// List of Strings.
FUNCTION_BLOCK FB_LongStringList
VAR
	List : ARRAY[ 0 .. GVL_List.LIST_SIZE - 1 ] OF LongString; // hold list
	_Count : UDINT := 0; // number of items.
END_VAR

// Add item to list. TRUE if successful. 
METHOD PUBLIC AddItem : BOOL
VAR_INPUT
	Item : LongString; // item to add.
END_VAR
IF _Count < GVL_List.LIST_SIZE THEN
	List[_Count] := Item; // list is zero indexed, so number of items points at next free space.
	_Count := _Count + 1; 
	AddItem := TRUE;
END_IF
END_METHOD

// Removes all list items
METHOD PUBLIC Clear
MEMSET(ADR(List[0]), 0, SIZEOF(List));
_Count := 0;
END_METHOD

// TRUE if Item is in FB_List.
METHOD PUBLIC Contains : BOOL
VAR_INPUT
	Item : LongString; // Item to check.
END_VAR
Contains := FindIndex(Item) >= 0;
END_METHOD

// TRUE if supplied key part is in any entry
METHOD PUBLIC ContainsPartial : BOOL
VAR_INPUT
	PartialItem : LongString;
END_VAR
ContainsPartial := FindIndexPartialKey(PartialItem) >= 0;
END_METHOD

METHOD CopyList
VAR_IN_OUT
	ListToCopyTo : ARRAY[ 0 .. GVL_List.LIST_SIZE - 1 ] OF LongString; // hold list
END_VAR
ListToCopyTo := THIS^.List;
END_METHOD

METHOD CopyListAndClear
VAR_IN_OUT
	ListToCopyTo : ARRAY[ 0 .. GVL_List.LIST_SIZE - 1 ] OF LongString; // hold list
END_VAR
THIS^.CopyList( ListToCopyTo );
THIS^.Clear();
END_METHOD

{attribute 'monitoring' := 'call'}
// Number of items in list.
PROPERTY PUBLIC Count : UDINT
GET
Count := _Count;
END_GET
END_PROPERTY

METHOD PUBLIC FindIndex : INT
VAR_INPUT
	Item : LongString; // Item to check.
END_VAR
VAR
	i : UINT := 0;
END_VAR
FindIndex := -1;
i := 0;
WHILE ( (FindIndex < 0) AND (i < _Count) ) DO
	
	FindIndex := SEL(Item = List[i], FindIndex, TO_INT(i) ); // if it matches, return the position.
	i := i + 1;
	
END_WHILE
END_METHOD

// Find first index where list entry contains supplied key.
METHOD PUBLIC FindIndexPartialKey : INT
VAR_INPUT
	PartialKey : LongString; // Item to check.
END_VAR
VAR
	i : UINT := 0;
END_VAR
FindIndexPartialKey := -1;
i := 0;
WHILE ( (FindIndexPartialKey < 0) AND (i < _Count) ) DO
	
	IF FIND(List[i],PartialKey) > 0 THEN
		FindIndexPartialKey := TO_INT(i);
	END_IF

	i := i + 1;
	
END_WHILE
END_METHOD

// Return item in list at index position. Returns empty string if invalid index.
METHOD PUBLIC GetIndex : LongString
VAR_INPUT
	Index : UDINT;
END_VAR
THIS^.TryGetIndex(Index,  GetIndex);
END_METHOD

//Remove the specified index. Shuffle remaining so list is intact.
METHOD PUBLIC RemoveIndex : BOOL
VAR_INPUT
	Index : UDINT;
END_VAR
IF Index >= _Count THEN // invalid index request.
	RETURN;
END_IF

IF Index < _Count - 1 THEN // If Index = _Count -1, last two lines sufficient.

	MEMMOVE( 
		destAddr := ADR( List[Index] ), 
		srcAddr := ADR( List[Index + 1] ), 
		n := SIZEOF(List[0]) * (_Count - Index - 1)
	);
	
END_IF

RemoveIndex := TRUE;

List[_Count - 1] := ''; // default the "old" end of the list.
_Count := _Count - 1; // reduce count.
END_METHOD

// TRUE if successful and list item in sItem
METHOD PUBLIC TryGetIndex : BOOL
VAR_INPUT
	Index : UDINT;
END_VAR
VAR_IN_OUT
	Item : LongString;
END_VAR
IF Index < _Count THEN
	TryGetIndex := TRUE;
	Item := List[Index];
END_IF
END_METHOD

END_FUNCTION_BLOCK

(* stored: Version 1.1.0.1, ProductVersion 3.1.4022.18
   POU FB_LongStringList: Id {6333a25e-a629-45cc-8282-40085d67c3f6}, SpecialFunc None
   Method AddItem: Id {cf250be8-a57e-4bea-aa0d-1037bf68190d}
   Method Clear: Id {97d94b3c-563f-4c5f-b952-456d7d913996}
   Method Contains: Id {72303850-6b2e-47a0-9b28-12bd5a42520d}
   Method ContainsPartial: Id {1938cd61-030a-4755-8a09-0ccff61e39c1}
   Method CopyList: Id {8b104ccb-382b-483e-ba85-1021b4e261da}
   Method CopyListAndClear: Id {486bfd6f-4bd8-4ffd-8dbd-2e418e677e6d}
   Property Count: Id {a8736c8b-aa4f-4638-afa9-3a2d623140c4}
   Get Get: Id {96b21c6b-3e47-4464-b4ca-d0ddec289dd9}
   Method FindIndex: Id {31ec6181-37e6-4510-900f-a9fd5567b870}
   Method FindIndexPartialKey: Id {4d772669-123e-4bf8-a1f9-c02b0cb772c6}
   Method GetIndex: Id {c1898d26-8b70-41ec-9579-3e585fe95301}
   Method RemoveIndex: Id {a7f9c6cc-277e-4084-b359-437c6f70b552}
   Method TryGetIndex: Id {c478a2dd-cf35-489b-bd56-1bf34db95e14} *)
